TYPE ST_ValveErrorList :
STRUCT 
	errOpenTimeout: 		STRING	:= 'alarm open timeout';
	errLostOpenPosition: 	STRING	:= 'lost open position';
	errCloseTimeout: 		STRING	:= 'alarm closing timeout';
	errLostClosePosition: 	STRING	:= 'lost close position';
	errBothSensorOn: 		STRING	:= 'alarm both sensor on';
END_STRUCT
END_TYPE

(* stored: Version 1.1.0.1, ProductVersion 3.1.4024.13
   DUT ST_ValveErrorList: Id {16a7da1a-b268-4d73-948a-5454623bf3a2} *)
